//Timeout and clear request
IF (tBPTMtimeout.Q) THEN
    fbArbiter.RemoveRequest(bptm.i_TransitionAssertionID);
    fbArbiter.RemoveRequest(bptm.i_nRequestedAssertionID);
END_IF
END_ACTION

METHOD PUBLIC M_IsClosed : BOOL
VAR_INPUT
END_VAR
M_IsClosed := (This^.iq_stValve.eState = E_ValvePositionState.CLOSED);
END_METHOD

METHOD PUBLIC M_IsOpen : BOOL
VAR_INPUT
END_VAR
M_IsOpen := (This^.iq_stValve.eState = E_ValvePositionState.OPEN);
END_METHOD

// Use this Methode to Open or close the valve by setting the OPN_SW to the input value.
METHOD PUBLIC M_Set_CLS_SW : BOOL
VAR_INPUT
        value:BOOL;
END_VAR
This^.iq_stValve.pv_xCLS_SW := value;
END_METHOD

END_FUNCTION_BLOCK
